SUBAPPLICATION Uebung_054 (* DigitalInput_I1-_I4 auf DigitalOutput_Q1-_Q4 *)
  (* Standard: 61499-2; Description: Copyright (c) 2023 Meisterschulen am Ostbahnhof This program and the accompanying materials are made available under the terms of the Eclipse Public License 2.0 which is available at https://www.eclipse.org/legal/epl-2.0/ SPDX-License-Identifier: EPL-2.0 *)
  (* Version 1.0, 2023-10-23, Franz Höpfinger, Meisterschulen am Ostbahnhof *)
  IMPORT logiBUS::io::DI::logiBUS_DI::Input_I1;
  IMPORT logiBUS::io::DI::logiBUS_DI::Input_I2;
  IMPORT logiBUS::io::DI::logiBUS_DI::Input_I3;
  IMPORT logiBUS::io::DI::logiBUS_DI::Input_I4;
  IMPORT logiBUS::io::DQ::logiBUS_DO::Output_Q1;
  IMPORT logiBUS::io::DQ::logiBUS_DO::Output_Q2;
  IMPORT logiBUS::io::DQ::logiBUS_DO::Output_Q3;
  IMPORT logiBUS::io::DQ::logiBUS_DO::Output_Q4;
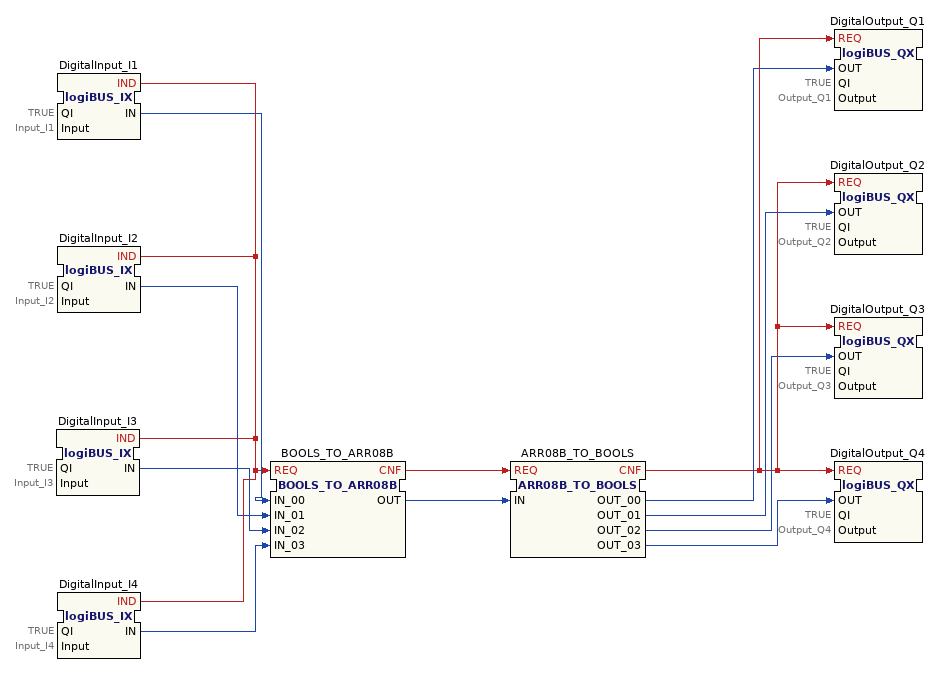
  FBS
    DigitalOutput_Q1 : logiBUS::io::DQ::logiBUS_QX(QI := TRUE, Output := Output_Q1);
    DigitalInput_I1 : logiBUS::io::DI::logiBUS_IX(QI := TRUE, Input := Input_I1);
    DigitalOutput_Q2 : logiBUS::io::DQ::logiBUS_QX(QI := TRUE, Output := Output_Q2);
    DigitalInput_I2 : logiBUS::io::DI::logiBUS_IX(QI := TRUE, Input := Input_I2);
    DigitalOutput_Q3 : logiBUS::io::DQ::logiBUS_QX(QI := TRUE, Output := Output_Q3);
    DigitalInput_I3 : logiBUS::io::DI::logiBUS_IX(QI := TRUE, Input := Input_I3);
    DigitalOutput_Q4 : logiBUS::io::DQ::logiBUS_QX(QI := TRUE, Output := Output_Q4);
    DigitalInput_I4 : logiBUS::io::DI::logiBUS_IX(QI := TRUE, Input := Input_I4);
    ARR08B_TO_BOOLS : ARR08B_TO_BOOLS;
    BOOLS_TO_ARR08B : BOOLS_TO_ARR08B;
  END_FBS
  EVENT_CONNECTIONS
    BOOLS_TO_ARR08B.CNF TO ARR08B_TO_BOOLS.REQ;
    DigitalInput_I1.IND TO BOOLS_TO_ARR08B.REQ;
    DigitalInput_I2.IND TO BOOLS_TO_ARR08B.REQ;
    DigitalInput_I3.IND TO BOOLS_TO_ARR08B.REQ;
    DigitalInput_I4.IND TO BOOLS_TO_ARR08B.REQ;
    ARR08B_TO_BOOLS.CNF TO DigitalOutput_Q1.REQ;
    ARR08B_TO_BOOLS.CNF TO DigitalOutput_Q2.REQ;
    ARR08B_TO_BOOLS.CNF TO DigitalOutput_Q3.REQ;
    ARR08B_TO_BOOLS.CNF TO DigitalOutput_Q4.REQ;
  END_CONNECTIONS
  DATA_CONNECTIONS
    BOOLS_TO_ARR08B.OUT TO ARR08B_TO_BOOLS.IN;
    DigitalInput_I1.IN TO BOOLS_TO_ARR08B.IN_00;
    DigitalInput_I2.IN TO BOOLS_TO_ARR08B.IN_01;
    DigitalInput_I3.IN TO BOOLS_TO_ARR08B.IN_02;
    DigitalInput_I4.IN TO BOOLS_TO_ARR08B.IN_03;
    ARR08B_TO_BOOLS.OUT_00 TO DigitalOutput_Q1.OUT;
    ARR08B_TO_BOOLS.OUT_01 TO DigitalOutput_Q2.OUT;
    ARR08B_TO_BOOLS.OUT_02 TO DigitalOutput_Q3.OUT;
    ARR08B_TO_BOOLS.OUT_03 TO DigitalOutput_Q4.OUT;
  END_CONNECTIONS
END_SUBAPPLICATION
